	DATA_BLOCK DB149
	TITLE =DBG049M  AERATION AIR STEEPING 9
	//COPYRIGHT:    (C) 2009  BUHLER AG, CH-9240 UZWIL, SWITZERLAND
	//
	//PRODUCT:      WinCoS_BIW01_09
	//
	//TITLE:        AERATION AIR STEEPING 9
	//                Machine group DB
	//                Maschinengruppen-DB
	//
	//-------------------------------------------------------------------------
	//
	//IDENT:        AUTHOR:             DEPT:             DATE:
	//
	//P01_DB149.1.0 K.Renz              CSB41             13.Jan.2010
	//              1st Release
	//
	//-------------------------------------------------------------------------
	//
	//PURPOSE:
	//
	//MANUAL :
	//
	//RESTRICTIONS:
	//
	//-------------------------------------------------------------------------
	AUTHOR  : KR
	FAMILY  : USW
	NAME    : DBG049M
	VERSION : 00.00

	FB149
	BEGIN
	      #Gr.Par.ParObjectNo 	:=4900;
	      #Gr.Par.ParIdling      	:=2;
	      #Gr.Par.ParMgr	        :=True;
	      #Gr.Par.ParWgr	        :=False;
	      #Gr.Par.ParGgr	        :=False;
	      #Gr.Par.ParEmptyingTime 	:=0;
	      #Gr.Par.ParHornCode       :=1;
	//Parameter =A-1119-QXV/BZS41/42 : AERATION AIR RING ST 9
	      #A_1119_QXV_BZS41_42.Par.ParObjectNo                             :=4901;
	      #A_1119_QXV_BZS41_42.Par.ParMsgType                              :=7081;
	      #A_1119_QXV_BZS41_42.Par.ParHornCode                             :=1;
	      #A_1119_QXV_BZS41_42.Par.ParMonTime                              :=100;
	      #A_1119_QXV_BZS41_42.Par.ParPulseTimeHN                          :=5;
	      #A_1119_QXV_BZS41_42.Par.ParPulseTimeLN                          :=5;
	      #A_1119_QXV_BZS41_42.Par.ParIdlingTime                           :=0;
	      #A_1119_QXV_BZS41_42.Par.ParDelayTime                            :=0;
	      #A_1119_QXV_BZS41_42.Par.ParLogOff                               :=False;
	      #A_1119_QXV_BZS41_42.Par.ParManual                               :=True;
	      #A_1119_QXV_BZS41_42.Par.ParPulseValve                           :=False;
	      #A_1119_QXV_BZS41_42.Par.ParContValve                            :=True;
	      #A_1119_QXV_BZS41_42.Par.ParManualFlap                           :=False;
	//
	//
	END_DATA_BLOCK
